SUBAPPLICATION page (* Subapplication Type *)
  (* Standard: 61499-2 *)
  (* Version 1.0, 2025-07-11, franz *)
  PACKAGE MyLib::sys::page;
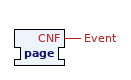
  EVENT_OUTPUT
    CNF; (* Execution Confirmation *)
  END_EVENT
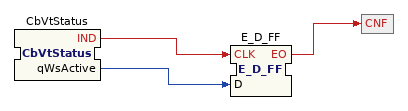
  FBS
    CbVtStatus : isobus::UT::status::CbVtStatus;
    E_D_FF : iec61499::events::E_D_FF;
  END_FBS
  EVENT_CONNECTIONS
    CbVtStatus.IND TO E_D_FF.CLK;
    E_D_FF.EO TO CNF;
  END_CONNECTIONS
  DATA_CONNECTIONS
    CbVtStatus.qWsActive TO E_D_FF.D;
  END_CONNECTIONS
END_SUBAPPLICATION
